TYPE ST_APP_STATE :
STRUCT
  AppInit             : E_PROGRESS;
  State            : E_INSTANCE_STATE;
END_STRUCT
END_TYPE

(* stored: Version 1.1.0.1
   DUT ST_APP_STATE: Id {b5b8f60b-c602-4356-8568-f704c7d8d195} *)
